(* LS Electric XG5000 project: library *)
(* PLC LSPLC *)

PROGRAM NewProgram (* task: 스캔 프로그램 *)
VAR
    FL : BOOL;
    INST : 오초깜빡이;
    NFL : BOOL;
    OFF : BOOL;
END_VAR

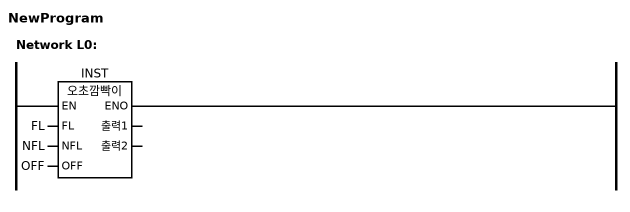
(* Rung L0 *)
INST(FL := FL, NFL := NFL, OFF := OFF);
END_PROGRAM